{attribute 'qualified_only'}
{attribute 'strict'}
{attribute 'to_string'}
TYPE E_MachineOpMode:
(
	AUTOMATIC,
    MANUAL
);
END_TYPE

(* stored: Version 1.1.0.1
   DUT E_MachineOpMode: Id {a6a73333-d32a-4c6d-abb3-0388e5a62438} *)
